TYPE ATV212 :
STRUCT
	fOutputFrequencyStatus	: REAL;
	fOutputCurrentStatus	: REAL;
	fOutputVoltageStatus	: REAL;
	fMotorSpeedStatus		: REAL;
END_STRUCT
END_TYPE

(* stored: Version 1.1.0.1, ProductVersion 3.1.4022.18
   DUT ATV212: Id {408cdde8-dbfa-4c19-8885-4e1f6d601963} *)
